{attribute 'qualified_only'}
VAR_GLOBAL
Bus : DUT_Busdiagnose;
END_VAR

(* stored: Version 1.1.0.1
   GVL GVL_Busdiagnose: Id {1c760060-1518-4826-af82-39d91bdbfa4e} *)
